Omron CX-Programmer project NewProject (CX-Programmer 9.75)

# PLC NewPLC1: CJ2M CPU11

## Global symbols (name address type ; comment)
1.00 BOOL  ; 100

## Program NewProgram1 (cyclic task 0)

### Section Section1

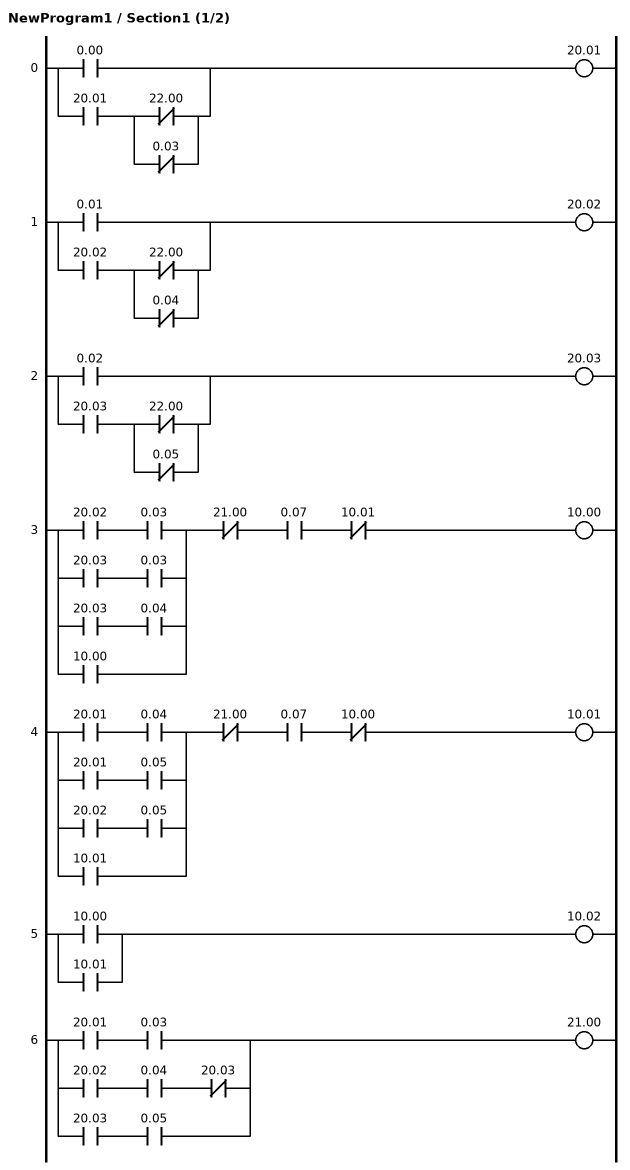
; rung 0
LD 0.00
LD 20.01
LDNOT 22.00
ORNOT 0.03
ANDLD
ORLD
OUT 20.01
; rung 1
LD 0.01
LD 20.02
LDNOT 22.00
ORNOT 0.04
ANDLD
ORLD
OUT 20.02
; rung 2
LD 0.02
LD 20.03
LDNOT 22.00
ORNOT 0.05
ANDLD
ORLD
OUT 20.03
; rung 3
LD 20.02
AND 0.03
LD 20.03
AND 0.03
ORLD
LD 20.03
AND 0.04
ORLD
OR 10.00
ANDNOT 21.00
AND 0.07
ANDNOT 10.01
OUT 10.00
; rung 4
LD 20.01
AND 0.04
LD 20.01
AND 0.05
ORLD
LD 20.02
AND 0.05
ORLD
OR 10.01
ANDNOT 21.00
AND 0.07
ANDNOT 10.00
OUT 10.01
; rung 5
LD 10.00
OR 10.01
OUT 10.02
; rung 6
LD 20.01
AND 0.03
LD 20.02
AND 0.04
ANDNOT 20.03
ORLD
LD 20.03
AND 0.05
ORLD
OUT 21.00

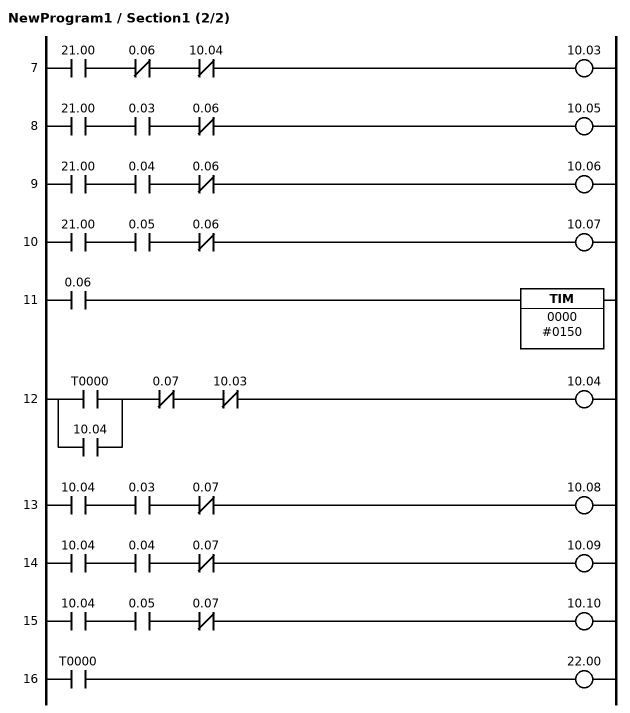
; rung 7
LD 21.00
ANDNOT 0.06
ANDNOT 10.04
OUT 10.03
; rung 8
LD 21.00
AND 0.03
ANDNOT 0.06
OUT 10.05
; rung 9
LD 21.00
AND 0.04
ANDNOT 0.06
OUT 10.06
; rung 10
LD 21.00
AND 0.05
ANDNOT 0.06
OUT 10.07
; rung 11
LD 0.06
TIM 0000 #0150
; rung 12
LD T0000
OR 10.04
ANDNOT 0.07
ANDNOT 10.03
OUT 10.04
; rung 13
LD 10.04
AND 0.03
ANDNOT 0.07
OUT 10.08
; rung 14
LD 10.04
AND 0.04
ANDNOT 0.07
OUT 10.09
; rung 15
LD 10.04
AND 0.05
ANDNOT 0.07
OUT 10.10
; rung 16
LD T0000
OUT 22.00

### Section END
; rung 0
END(001)